PROGRAM PRG1_Conveyer_Operation
VAR
END_VAR


// bereken snelheid

GVL.ladingGewicht := GVL.weegcelWaarde;									
GVL.geschrevenSnelheid := FC1_Bereken_Snelheid(GVL.ladingGewicht);

END_PROGRAM

(* stored: Version 1.1.0.1, ProductVersion 3.1.4024.12
   POU PRG1_Conveyer_Operation: Id {45b7ed08-ad47-4fa3-b041-11199023376c}, SpecialFunc None *)
